FUNCTION_BLOCK EH_TimeOut (* Basic FB with empty ECC *)
  (* Standard: 61499-2 *)
  (* Version 1.0, 2020-07-27, dummy *)
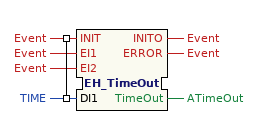
  EVENT_INPUT
    INIT WITH DI1;
    EI1;
    EI2;
  END_EVENT
  EVENT_OUTPUT
    INITO;
    ERROR;
  END_EVENT
  VAR_INPUT
    DI1 : TIME;
  END_VAR
  PLUGS
    TimeOut : ATimeOut;
  END_PLUGS
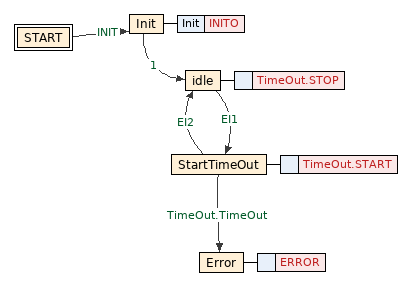
  EC_STATES
    START; (* Initial State *)
    Init : Init -> INITO;
    idle : -> TimeOut.STOP;
    StartTimeOut : -> TimeOut.START;
    Error : -> ERROR;
  END_STATES
  EC_TRANSITIONS
    START TO Init := INIT;
    Init TO idle := 1;
    idle TO StartTimeOut := EI1;
    StartTimeOut TO Error := TimeOut.TimeOut;
    StartTimeOut TO idle := EI2;
  END_TRANSITIONS
  ALGORITHM Init IN ST:
TimeOut.DT := DI1;
  END_ALGORITHM
END_FUNCTION_BLOCK
